TYPE E_DeviceEndianness :
(
	LittleEndian,
	BigEndian
);
END_TYPE

(* stored: Version 1.1.0.1, ProductVersion 3.1.4024.15
   DUT E_DeviceEndianness: Id {8c6a36e8-f33d-428b-b83a-481b140c04eb} *)
